FUNCTION_BLOCK SL_Stopper (* Stopper contract: Requires NeedleUp AND VialPresent AND (FilledMl > 0.0) AND NOT Stoppered; Ensures Stoppered; Invariant NeedleUp AND VialPresent *)
  (* Standard: 61499-2 *)
  (* Version 2.0, 2026-09-27, Project contributors, Filling cell reference model *)
  PACKAGE fillingcell;
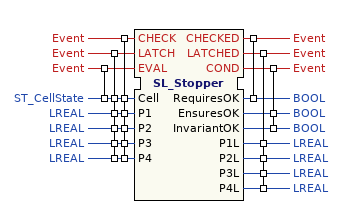
  EVENT_INPUT
    CHECK WITH Cell, P1, P2, P3, P4;
    LATCH WITH Cell, P1, P2, P3, P4;
    EVAL WITH Cell;
  END_EVENT
  EVENT_OUTPUT
    CHECKED WITH RequiresOK;
    LATCHED WITH P1L, P2L, P3L, P4L;
    COND WITH EnsuresOK, InvariantOK;
  END_EVENT
  VAR_INPUT
    Cell : fillingcell::ST_CellState;
    P1 : LREAL;
    P2 : LREAL;
    P3 : LREAL;
    P4 : LREAL;
  END_VAR
  VAR_OUTPUT
    RequiresOK : BOOL;
    EnsuresOK : BOOL;
    InvariantOK : BOOL;
    P1L : LREAL;
    P2L : LREAL;
    P3L : LREAL;
    P4L : LREAL;
  END_VAR
  EC_STATES
    CHECK : CHECK -> CHECKED;
    LATCH : LATCH -> LATCHED;
    EVAL : EVAL -> COND;
  END_STATES
  ALGORITHM CHECK IN ST:
RequiresOK := Cell.Valid AND Cell.Safe AND (Cell.NeedleUp AND Cell.VialPresent AND (Cell.FilledMl > 0.0) AND NOT Cell.Stoppered);
  END_ALGORITHM
  ALGORITHM LATCH IN ST:
P1L := P1;
P2L := P2;
P3L := P3;
P4L := P4;
  END_ALGORITHM
  ALGORITHM EVAL IN ST:
EnsuresOK := Cell.Stoppered;
InvariantOK := Cell.Valid AND Cell.Safe AND (Cell.NeedleUp AND Cell.VialPresent);
  END_ALGORITHM
END_FUNCTION_BLOCK
